// TwinCAT 3 PLC project DataFluxPLC
// ProgramVersion: 3.1.4026.22
// libraries:
//   Tc2_Standard, * (Beckhoff Automation GmbH)
//   Tc2_System, * (Beckhoff Automation GmbH)
// project tree:
//   GVLs/ MachineData.TcGVL
//   / PlcTask.TcTTO
//   POUs/ ConveyorMain.TcPOU, MAIN.TcPOU, MotorControl.TcPOU
// real-time tasks:
//   TASK PlcTask: cycle T#10ms, priority 20, ADS port 350

CONFIGURATION DataFluxPLC
    RESOURCE PLC ON TwinCAT3
        TASK PlcTask(INTERVAL := T#10ms, PRIORITY := 20);
        PROGRAM MAIN WITH PlcTask : MAIN;
    END_RESOURCE
END_CONFIGURATION

// ---- GVLs/MachineData.TcGVL
{attribute 'qualified_only'}
VAR_GLOBAL
    ConveyorRunning : BOOL   := FALSE;
    MotorTemp       : REAL   := 72.5;
    PartCount       : INT    := 0;
END_VAR

// ---- POUs/MAIN.TcPOU
PROGRAM MAIN
VAR
    CycleTimer : TON;
END_VAR

CycleTimer(IN := NOT CycleTimer.Q, PT := T#1S);

IF CycleTimer.Q THEN
    MachineData.PartCount := MachineData.PartCount + 1;
    MachineData.MotorTemp       := MachineData.MotorTemp + 0.1;
    MachineData.ConveyorRunning := TRUE;
END_IF

END_PROGRAM

// ---- POUs/ConveyorMain.TcPOU
FUNCTION_BLOCK ConveyorMain
VAR_INPUT
    Start       : BOOL;
    Stop        : BOOL;
    FaultReset  : BOOL;
END_VAR
VAR_OUTPUT
    Running     : BOOL;
    Faulted     : BOOL;
END_VAR
VAR
    RunningInternal : BOOL;
END_VAR


IF FaultReset THEN
    Faulted := FALSE;
END_IF

IF Start AND NOT Faulted THEN
    RunningInternal := TRUE;
END_IF

IF Stop THEN
    RunningInternal := FALSE;
END_IF

Running := RunningInternal;

END_FUNCTION_BLOCK

// ---- POUs/MotorControl.TcPOU
FUNCTION_BLOCK MotorControl
VAR_INPUT
END_VAR
VAR_OUTPUT
END_VAR
VAR
END_VAR

END_FUNCTION_BLOCK
